PROGRAM main
  VAR_INPUT
    X0 : BOOL;
    X1 : BOOL;
    X2 : BOOL;
  END_VAR
  VAR_OUTPUT
    Y0 : BOOL;
  END_VAR
  VAR
    M0 : BOOL;
  END_VAR

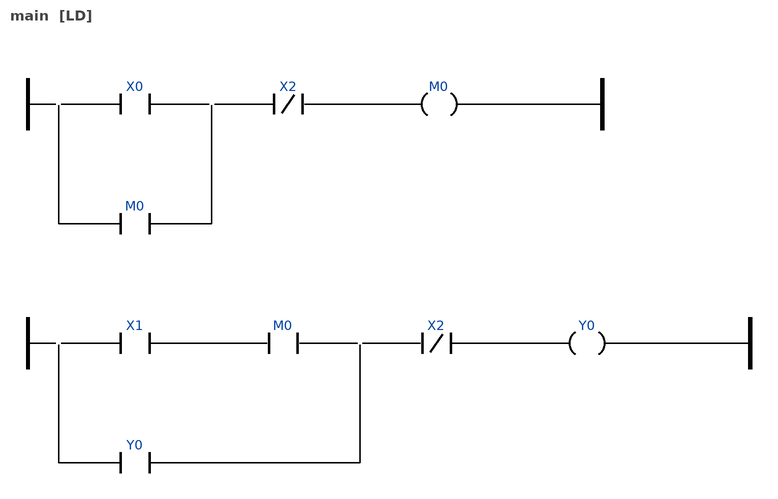
(* LD diagram, written out as Structured Text *)
M0 := (X0 OR M0) AND NOT X2;
Y0 := (Y0 OR X1 AND M0) AND NOT X2;
END_PROGRAM
